// TIA Portal project "1500连接abb" (V16)

(* hardware
DEVICE "S71500/ET200MP station_1"  S7-1500 station
   slot 0: "导轨_0"  Rack  6ES7 590-1***0-0AA0
   slot 1: "PLC_1"  CPU 1515-2 PN  6ES7 515-2AM02-0AB0  V2.8
      slot 3: "CPU 显示_1"  6ES7591-1BA00-0AA0
      slot 32768: "PROFINET 接口_1"  X1
         slot 32769: "端口_1"  X1 P1
         slot 32770: "端口_2"  X1 P2
      slot 33024: "PROFINET 接口_2"  X2
         slot 33025: "端口_1"  X2 P1
      slot 34817: "Virtual CP interface port_1"  Virtual CP interface port  Virtual CP interface port
*)

// ===== PLC "PLC_1"  CPU 1515-2 PN =====

VAR_GLOBAL   // PLC tag table "IO表"
   "启动运输带" AT %Q0.0 : Bool;
   "夹取" AT %Q0.1 : Bool;
   "放开" AT %Q0.2 : Bool;
   "开门" AT %Q0.3 : Bool;
   "关门" AT %Q0.4 : Bool;
   "推杆" AT %Q0.5 : Bool;
   "收杆" AT %Q0.6 : Bool;
   "传感器1" AT %I0.0 : Bool;
   "传感器2" AT %I0.1 : Bool;
   "传感器3" AT %I0.2 : Bool;
   "传感器4" AT %I0.3 : Bool;
   "传感器5" AT %I0.4 : Bool;
   "传感器6" AT %I0.5 : Bool;
   "传感器7" AT %I0.6 : Bool;
   "传感器8" AT %I0.7 : Bool;
   "传感器9" AT %I1.0 : Bool;
   "启动" AT %M0.0 : Bool;
   "停止" AT %M0.1 : Bool;
   "绿灯" AT %M0.2 : Bool;
   "黄灯" AT %M0.3 : Bool;
   "红灯" AT %M0.4 : Bool;
END_VAR

ORGANIZATION_BLOCK "Main"   // OB1, LAD, ProgramCycle
TITLE = "Main Program Sweep (Cycle)"
{ S7_Optimized_Access := 'TRUE' }
VERSION : 0.1
   VAR_INPUT
      Initial_Call : Bool;   // Initial call of this OB
      Remanence : Bool;   // =True, if remanent data are available
   END_VAR
BEGIN

REGION Network 1: 启动传送带
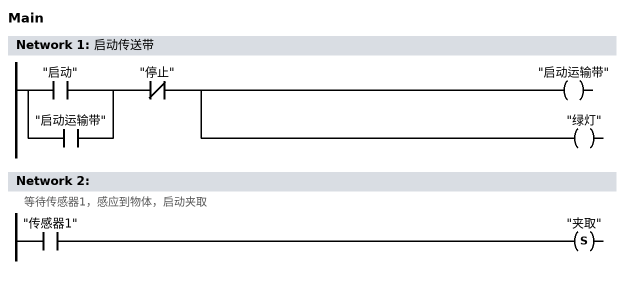
   RUNG wire#powerrail
      Contact( "启动" )
      wire#w1
      I_Contact( "停止" )
      wire#w2
      Coil( "启动运输带" )
   END_RUNG
   RUNG wire#powerrail
      Contact( "启动运输带" )
   END_RUNG wire#w1
   RUNG wire#w2
      Coil( "绿灯" )
   END_RUNG
   // the same network as SCL:
   "启动运输带" := ("启动" OR "启动运输带") AND NOT "停止";
   "绿灯" := "启动运输带";
END_REGION

REGION Network 2
   // 等待传感器1，感应到物体，启动夹取
   RUNG wire#powerrail
      Contact( "传感器1" )
      S_Coil( "夹取" )
   END_RUNG
   // the same network as SCL:
   IF "传感器1" THEN "夹取" := TRUE; END_IF;
END_REGION
END_ORGANIZATION_BLOCK